// TIA Portal V20 export
DATA_BLOCK "PM8"   // DB282
// stored: MemoryReserve 100
   VAR
      "HIPOT TAB CONTACTOR FORWARD" : Bool;
      "HIPOT TAB CONTACTOR BACKWARD" : Bool;
      "HIPOT TAB CONTACTOR LEFT CLOSE" : Bool;
      "HIPOT TAB CONTACTOR LEFT OPEN" : Bool;
      "HIPOT TAB CONTACTOR RIGHT CLOSE" : Bool;
      "HIPOT TAB CONTACTOR RIGHT OPEN" : Bool;
      SPARE : Bool;
      SPARE_1 : Bool;
      SPARE_2 : Bool;
      SPARE_3 : Bool;
      "HIPOT & THICKNESS STAGE LIFT FRONT UP" : Bool;
      "HIPOT & THICKNESS STAGE LIFT FRONT DOWN" : Bool;
      "HIPOT & THICKNESS STAGE LIFT REAR UP" : Bool;
      "HIPOT & THICKNESS STAGE LIFT REAR DOWN" : Bool;
      SPARE_4 : Bool;
      SPARE_5 : Bool;
   END_VAR
BEGIN
END_DATA_BLOCK
